// TIA Portal V18 export
TYPE "UDT_AHUsState"
// stored: IsFailsafeCompliant false
   STRUCT
      cPreviousOne : Array[1..3] of Byte;
      cActual : Array[1..3] of Byte;
      cTarget : Array[1..3] of Byte;
      xActualStateEdge : Array[1..3] of Bool;
      cSimpleForHMI : Array[1..3] of Byte;
      iCounterOfSwitchingBtwActualStates : Array[1..3] of Int;
   END_STRUCT;
   // // cSimpleForHMI[1] : 0 - Not Exist, 1-Stopped, 1- Run, 2 - Alarm Blocked
   // // cSimpleForHMI[2] : 0 - Not Exist, 1-Stopped, 1- Run, 2 - Alarm Blocked
   // // cSimpleForHMI[3] : 0 - Not Exist, 1-Stopped, 1- Run, 2 - Alarm Blocked
END_TYPE
